FUNCTION_BLOCK FB_HomeDirect
VAR_INPUT
    En: BOOL;
    bReset: BOOL;
    bExecute: BOOL;
    fHomePosition:LREAL;
END_VAR
VAR_IN_OUT
    Axis: AXIS_REF;
END_VAR
VAR_OUTPUT
    EnO: BOOL;
    bBusy: BOOL;
    bDone: BOOL;
    bHomed:BOOL;
    bError: BOOL;
    nErrorId: UDINT;
END_VAR
VAR
    fbHome: MC_Home;
END_VAR

En:=EnO;
IF bReset THEN
    bError:=FALSE;
    nErrorId:=0;
END_IF

fbHome(
    Execute:=bExecute,
    Position:=fHomePosition,
    HomingMode:=MC_Direct,
    bCalibrationCam:=FALSE,
    Axis:=Axis
    );

bBusy:=fbHome.Busy;
bDone:=fbHome.Done;
bHomed:=Axis.Status.Homed;

bError:=fbHome.Error;

IF fbHome.Error THEN
  nErrorId:=fbHome.ErrorID;
END_IF

END_FUNCTION_BLOCK

(* stored: Version 1.1.0.1, ProductVersion 3.1.4024.0
   POU FB_HomeDirect: Id {bcba1819-aaef-4ffc-bcb6-e637240bf3e1}, SpecialFunc None *)
